INTERFACE I_NodePrototype EXTENDS I_Disposable

METHOD PUBLIC Accept
VAR_INPUT
	Visitor : I_NodePrototypeVisitor;
END_VAR
END_METHOD

METHOD PUBLIC Clone : I_Node
VAR_INPUT
END_VAR
END_METHOD

PROPERTY PUBLIC Node : I_Node
GET
END_GET
END_PROPERTY

PROPERTY PUBLIC Path : T_MAXSTRING
GET
END_GET
END_PROPERTY

END_INTERFACE

(* stored: Version 1.1.0.1, ProductVersion 3.1.4024.12
   Itf I_NodePrototype: Id {bdb453bc-5a57-421d-b123-ac91467b8c03}
   Method Accept: Id {366fd43a-bff6-43ac-ad51-46889d5e807e}
   Method Clone: Id {440e2f18-cc78-4552-ae6b-502e6b3008ae}
   Property Node: Id {b3045315-d1b5-4d5e-a05c-1072061948db}
   Get Get: Id {52768432-d8f6-420b-8bb3-8857014f1fe7}
   Property Path: Id {3a017e7f-53d6-4af2-9231-348f9d24272f}
   Get Get: Id {b8fbeff6-25a9-4713-bf4b-df5493516c3c} *)
